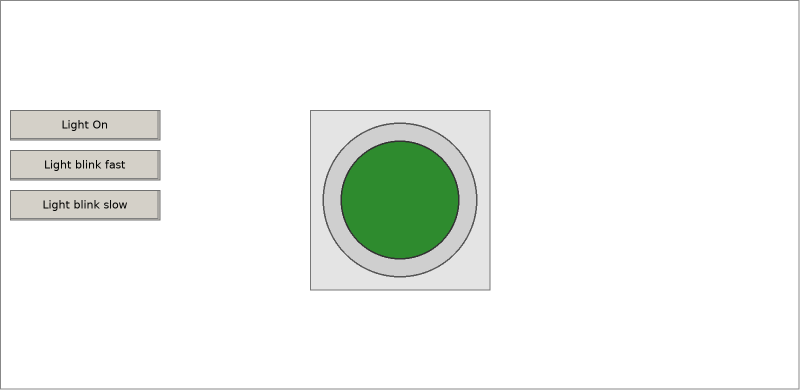
VISUALIZATION VisuPushbuttonLightControl  // 800x390
VAR_IN_OUT
	fbManualControler	: FB_ManualController ;
END_VAR
    PushSwitch (310,110 180x180), variable: fbManualControler.pDevPBL^.bFcoInputActive, behaviour: TOGGLE, style: Switch-PushSwitch-Green
    Button (10,110 150x30), "Light On"
        toggle fbManualControler.pDevPBL^.fbLight.bCmdOn
    Button (10,150 150x30), "Light blink fast"
        toggle fbManualControler.pDevPBL^.fbLight.bCmdBlinkFast
    Button (10,190 150x30), "Light blink slow"
        toggle fbManualControler.pDevPBL^.fbLight.bCmdBlinkSlow
END_VISUALIZATION

(* stored: Version 1.1.0.1, ProductVersion 3.1.4024.11
   Visu VisuPushbuttonLightControl: Id {906eb558-e84d-0863-189b-a7ddcd3cb86b} *)
